PROGRAM p00_true_false
VAR
	M0: BOOL;
	M1: BOOL;
	S0: BOOL;
	L0: BOOL;
	S1: BOOL;
	L1: BOOL;
	L2: BOOL;
END_VAR

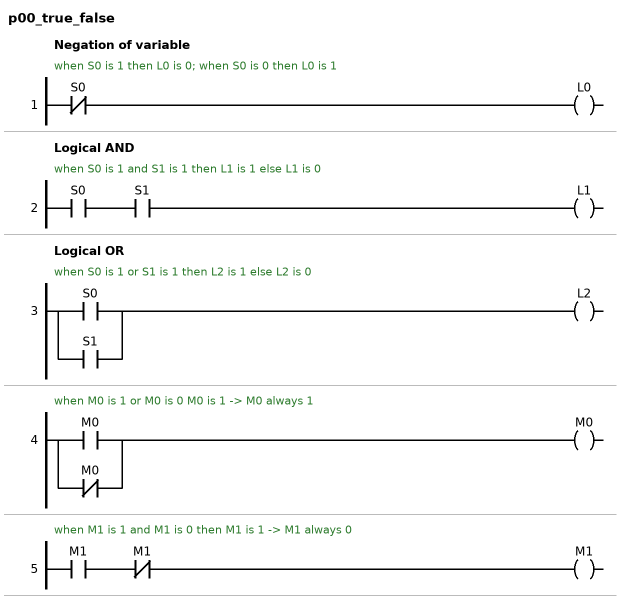
// NETWORK 1: Negation of variable
// when S0 is 1 then L0 is 0; when S0 is 0 then L0 is 1
L0 := NOT S0;

// NETWORK 2: Logical AND
// when S0 is 1 and S1 is 1 then L1 is 1 else L1 is 0
L1 := S0 AND S1;

// NETWORK 3: Logical OR
// when S0 is 1 or S1 is 1 then L2 is 1 else L2 is 0
L2 := S0 OR S1;

// NETWORK 4
// when M0 is 1 or M0 is 0 M0 is 1 -> M0 always 1
M0 := M0 OR NOT M0;

// NETWORK 5
// when M1 is 1 and M1 is 0 then M1 is 1 -> M1 always 0
M1 := M1 AND NOT M1;

END_PROGRAM

(* stored: Version 1.1.0.1, ProductVersion 3.1.4024.13
   POU p00_true_false: Id {daf84d60-9dea-4523-935e-4e1045f732ed}, SpecialFunc None *)
